FUNCTION_BLOCK FB_ConfigControl
VAR_INPUT
	a_pFBConfigJson : POINTER TO POINTER TO FB_ConfigBase; //pointer to pointer is an array
	ua_pFBConfigJson : UDINT;
END_VAR
VAR_OUTPUT
END_VAR
VAR
	fbRecipeJson : FB_ValuesJson;
	fbSystemJson : FB_ValuesJson;
	fbIOJson : FB_ValuesJson;
	fbAxisJson : FB_NCAxisJson_V2;
END_VAR

METHOD PUBLIC M_GetJsonAxis : HResult
VAR_INPUT
	lastResult : HRESULT;
END_VAR
VAR_IN_OUT
	pDoc : STRING(50000);
END_VAR
VAR CONSTANT
	uSizeOfStAnyType : UDINT := SIZEOF(PVOID);
END_VAR
VAR_INST
	uSizeOfArray : DINT;
	x : DINT;
	pFBConfigJson : POINTER TO POINTER TO FB_ConfigBase;	
	_fbResult : FB_ResultHelper_V2;
	pResult : POINTER TO HRESULT;
END_VAR
IF _fbResult.M_MethodResult(M_GetJsonAxis,ADR(pResult),lastResult) = FALSE THEN
	RETURN;
END_IF

uSizeOfArray := ua_pFBConfigJson/uSizeOfStAnyType - 1; //get number of items in array

fbAxisJson.ParseDocument(pDoc);
fbAxisJson.M_PraseSchemaJson();
FOR x := 0 TO uSizeOfArray BY 1 DO
	pFBConfigJson := a_pFBConfigJson + uSizeOfStAnyType*x;
	lastResult := pFBConfigJson^^.F_AXIS(lastResult,fbAxisJson.P_sJsonValues.jsonValue,ADR(fbAxisJson),TRUE);
END_FOR

fbAxisJson.CopyDocument(pDoc,SIZEOF(pDoc));
END_METHOD

METHOD PUBLIC M_GetJsonIO : HResult
VAR_INPUT
	lastResult : HRESULT;
END_VAR
VAR_IN_OUT
	pDoc : STRING(50000);
END_VAR
VAR CONSTANT
	uSizeOfStAnyType : UDINT := SIZEOF(PVOID);
END_VAR
VAR_INST
	uSizeOfArray : DINT;
	x : DINT;
	pFBConfigJson : POINTER TO POINTER TO FB_ConfigBase;	
	_fbResult : FB_ResultHelper_V2;
	pResult : POINTER TO HRESULT;
END_VAR
IF _fbResult.M_MethodResult(M_GetJsonIO,ADR(pResult),lastResult) = FALSE THEN
	RETURN;
END_IF


uSizeOfArray := ua_pFBConfigJson/uSizeOfStAnyType - 1; //get number of items in array


fbIOJson.M_CreateSchemaJson();
FOR x := 0 TO uSizeOfArray BY 1 DO
	pFBConfigJson := a_pFBConfigJson + uSizeOfStAnyType*x;
	lastResult := pFBConfigJson^^.F_IO(lastResult,fbIOJson.P_sJsonValues.jsonValue,ADR(fbIOJson),FALSE);
END_FOR


fbIOJson.CopyDocument(pDoc,SIZEOF(pDoc));
END_METHOD

METHOD PUBLIC M_GetJsonRecipe : HResult
VAR_INPUT
	lastResult : HRESULT;
END_VAR
VAR_IN_OUT
	pDoc : STRING(10000);
END_VAR

VAR CONSTANT
	uSizeOfStAnyType : UDINT := SIZEOF(PVOID);
END_VAR

VAR_INST
	bGet : BOOL;
	uSizeOfArray : DINT;
	x : DINT;
	pFBConfigJson : POINTER TO POINTER TO FB_ConfigBase;	
	_fbResult : FB_ResultHelper_V2;
	pResult : POINTER TO HRESULT;
END_VAR
IF _fbResult.M_MethodResult(M_GetJsonRecipe,ADR(pResult),lastResult) = FALSE THEN
	RETURN;
END_IF

uSizeOfArray := ua_pFBConfigJson/uSizeOfStAnyType - 1; //get number of items in array

fbRecipeJson.M_PraseSchemaJson();
FOR x := 0 TO uSizeOfArray BY 1 DO
	pFBConfigJson := a_pFBConfigJson + uSizeOfStAnyType*x;
	lastResult := pFBConfigJson^^.F_Recipe(lastResult,fbRecipeJson.P_sJsonValues.jsonValue,ADR(fbRecipeJson),TRUE);
END_FOR

fbRecipeJson.CopyDocument(pDoc,SIZEOF(pDoc));
END_METHOD

METHOD PUBLIC M_GetJsonSystem : HResult
VAR_INPUT
	lastResult : HRESULT;
END_VAR
VAR_IN_OUT
	pDoc : STRING(50000);
END_VAR
VAR CONSTANT
	uSizeOfStAnyType : UDINT := SIZEOF(PVOID);
END_VAR
VAR_INST
	uSizeOfArray : DINT;
	x : DINT;
	pFBConfigJson : POINTER TO POINTER TO FB_ConfigBase;	
	_fbResult : FB_ResultHelper_V2;
	pResult : POINTER TO HRESULT;
END_VAR
IF _fbResult.M_MethodResult(M_GetJsonSystem,ADR(pResult),lastResult) = FALSE THEN
	RETURN;
END_IF

uSizeOfArray := ua_pFBConfigJson/uSizeOfStAnyType - 1; //get number of items in array


fbSystemJson.M_CreateSchemaJson();
FOR x := 0 TO uSizeOfArray BY 1 DO
	pFBConfigJson := a_pFBConfigJson + uSizeOfStAnyType*x;
	lastResult := pFBConfigJson^^.F_System(lastResult,fbSystemJson.P_sJsonValues.jsonValue,ADR(fbSystemJson),TRUE);
END_FOR

fbSystemJson.CopyDocument(pDoc,SIZEOF(pDoc));
END_METHOD

METHOD PUBLIC M_SetJsonAxis : HResult
VAR_INPUT
	lastResult : HRESULT;
END_VAR
VAR_IN_OUT
	pDoc : STRING(50000);
END_VAR
VAR CONSTANT
	uSizeOfStAnyType : UDINT := SIZEOF(PVOID);
END_VAR
VAR_INST
	uSizeOfArray : DINT;
	x : DINT;
	pFBConfigJson : POINTER TO POINTER TO FB_ConfigBase;	
	_fbResult : FB_ResultHelper_V2;
	pResult : POINTER TO HRESULT;
END_VAR
IF _fbResult.M_MethodResult(M_SetJsonAxis,ADR(pResult),lastResult) = FALSE THEN
	RETURN;
END_IF

uSizeOfArray := ua_pFBConfigJson/uSizeOfStAnyType - 1; //get number of items in array


fbAxisJson.M_CreateSchemaJson();
FOR x := 0 TO uSizeOfArray BY 1 DO
	pFBConfigJson := a_pFBConfigJson + uSizeOfStAnyType*x;
	lastResult := pFBConfigJson^^.F_AXIS(lastResult,fbAxisJson.P_sJsonValues.jsonValue,ADR(fbAxisJson),TRUE);
END_FOR

fbAxisJson.CopyDocument(pDoc,SIZEOF(pDoc));
END_METHOD

METHOD PUBLIC M_SetJsonIO : HResult
VAR_INPUT
	lastResult : HRESULT;
END_VAR
VAR_IN_OUT
	pDoc : STRING(50000);
END_VAR
VAR CONSTANT
	uSizeOfStAnyType : UDINT := SIZEOF(PVOID);
END_VAR
VAR_INST
	uSizeOfArray : DINT;
	x : DINT;
	pFBConfigJson : POINTER TO POINTER TO FB_ConfigBase;	
	_fbResult : FB_ResultHelper_V2;
	pResult : POINTER TO HRESULT;
END_VAR
IF _fbResult.M_MethodResult(M_SetJsonIO,ADR(pResult),lastResult) = FALSE THEN
	RETURN;
END_IF

uSizeOfArray := ua_pFBConfigJson/uSizeOfStAnyType - 1; //get number of items in array


fbIOJson.M_CreateSchemaJson();
FOR x := 0 TO uSizeOfArray BY 1 DO
	pFBConfigJson := a_pFBConfigJson + uSizeOfStAnyType*x;
	lastResult := pFBConfigJson^^.F_IO(lastResult,fbIOJson.P_sJsonValues.jsonValue,ADR(fbIOJson),TRUE);
END_FOR


fbIOJson.CopyDocument(pDoc,SIZEOF(pDoc));
END_METHOD

METHOD PUBLIC M_SetJsonRecipe : HResult
VAR_INPUT
	lastResult : HRESULT;
END_VAR
VAR_IN_OUT
	pDoc : STRING(10000);
END_VAR

VAR CONSTANT
	uSizeOfStAnyType : UDINT := SIZEOF(PVOID);
END_VAR

VAR_INST
	bGet : BOOL;
	uSizeOfArray : DINT;
	x : DINT;
	pFBConfigJson : POINTER TO POINTER TO FB_ConfigBase;	
	_fbResult : FB_ResultHelper_V2;
	pResult : POINTER TO HRESULT;
END_VAR
IF _fbResult.M_MethodResult(M_SetJsonRecipe,ADR(pResult),lastResult) = FALSE THEN
	RETURN;
END_IF

uSizeOfArray := ua_pFBConfigJson/uSizeOfStAnyType - 1; //get number of items in array

fbRecipeJson.M_CreateSchemaJson();
FOR x := 0 TO uSizeOfArray BY 1 DO
	pFBConfigJson := a_pFBConfigJson + uSizeOfStAnyType*x;
	lastResult := pFBConfigJson^^.F_Recipe(lastResult,fbRecipeJson.P_sJsonValues.jsonValue,ADR(fbRecipeJson),FALSE);
END_FOR

fbRecipeJson.CopyDocument(pDoc,SIZEOF(pDoc));
END_METHOD

METHOD PUBLIC M_SetJsonSystem : HResult
VAR_INPUT
	lastResult : HRESULT;
END_VAR
VAR_IN_OUT
	pDoc : STRING(50000);
END_VAR
VAR CONSTANT
	uSizeOfStAnyType : UDINT := SIZEOF(PVOID);
END_VAR
VAR_INST
	uSizeOfArray : DINT;
	x : DINT;
	pFBConfigJson : POINTER TO POINTER TO FB_ConfigBase;	
	_fbResult : FB_ResultHelper_V2;
	pResult : POINTER TO HRESULT;
END_VAR
IF _fbResult.M_MethodResult(M_SetJsonSystem,ADR(pResult),lastResult) = FALSE THEN
	RETURN;
END_IF

uSizeOfArray := ua_pFBConfigJson/uSizeOfStAnyType - 1; //get number of items in array


fbSystemJson.M_CreateSchemaJson();
FOR x := 0 TO uSizeOfArray BY 1 DO
	pFBConfigJson := a_pFBConfigJson + uSizeOfStAnyType*x;
	lastResult := pFBConfigJson^^.F_System(lastResult,fbSystemJson.P_sJsonValues.jsonValue,ADR(fbSystemJson),FALSE);
END_FOR

fbSystemJson.CopyDocument(pDoc,SIZEOF(pDoc));
END_METHOD

END_FUNCTION_BLOCK

(* stored: Version 1.1.0.1, ProductVersion 3.1.4024.12
   POU FB_ConfigControl: Id {40efb18b-3f60-4fa1-aa5b-c43795a06346}, SpecialFunc None
   Method M_GetJsonAxis: Id {f2577cc8-ada7-4485-9fbd-d7c81979f777}
   Method M_GetJsonIO: Id {24d8351e-c4e8-46a7-988d-494288c63118}
   Method M_GetJsonRecipe: Id {46911a91-a1d5-4cf5-9cc2-9e277e00fa45}
   Method M_GetJsonSystem: Id {0b5fb081-6907-4da7-8fc5-e52fd4f1db29}
   Method M_SetJsonAxis: Id {765762fc-ea43-4377-89d7-628b8a9bb1cb}
   Method M_SetJsonIO: Id {132bf0dc-f494-4655-8dce-d202cd22afc3}
   Method M_SetJsonRecipe: Id {bfd8563a-59ab-4c37-958b-6beb44e7770e}
   Method M_SetJsonSystem: Id {aa4bbf75-637c-4be0-bbe1-fa1addb2eb27} *)
